// TIA Portal V20 export
// export: Created 2025-12-01T14:56:16.9516527Z, ExportSetting None, DisplayName Totally Integrated Automation Portal, DisplayVersion V20 Update 3, DisplayName TIA Portal Openness, DisplayVersion V20 Update 3, DisplayName TIA Portal Version Control Interface, DisplayVersion V20 Update 3, DisplayName STEP 7 Professional, DisplayVersion V20 Update 3, DisplayName STEP 7 Safety, DisplayVersion V20 Update 2, DisplayName WinCC Basic/Comfort/Advanced, DisplayVersion V20 Update 3, DisplayName WinCC Professional, DisplayVersion V20 Update 3, DisplayName WinCC Unified, DisplayVersion V20 Update 3
TYPE "UDT_Interlock_STV"
   STRUCT
      Load_arrival : Bool;
      LoadComplete : Bool;
      Load_ok : Bool;
      "Byte0.bit3" : Bool;
      "Byte0.bit4" : Bool;
      "Byte0.bit5" : Bool;
      "Byte0.bit6" : Bool;
      "Byte0.bit7" : Bool;
      Unload_Arrival : Bool;
      Unload_ok : Bool;
      UnloadComplete : Bool;
      Byte1_bit3 : Bool;
      Byte1_bit4 : Bool;
      Byte1_bit5 : Bool;
      Byte1_bit6 : Bool;
      Byte1_bit7 : Bool;
      Byte2_bit0 : Bool;
      Byte2_bit1 : Bool;
      Byte2_bit2 : Bool;
      Byte2_bit3 : Bool;
      Byte2_bit4 : Bool;
      Byte2_bit5 : Bool;
      Byte2_bit6 : Bool;
      Byte2_bit7 : Bool;
      Byte3_bit0 : Bool;
      Byte3_bit1 : Bool;
      Byte3_bit2 : Bool;
      Byte3_bit3 : Bool;
      Byte3_bit4 : Bool;
      Byte3_bit5 : Bool;
      Byte3_bit6 : Bool;
      Byte3_bit7 : Bool;
   END_STRUCT;
END_TYPE
